FUNCTION_BLOCK TelemetryRelativeHumidities EXTENDS SM_TelemetryRelativeHumidities
VAR_INPUT
END_VAR
VAR_OUTPUT
END_VAR
VAR
    _testVar_TelemetryRelativeHumidities : BOOL;
END_VAR

SUPER^(config := config);

END_FUNCTION_BLOCK

(* stored: Version 1.1.0.1, ProductVersion 3.1.0.36
   POU TelemetryRelativeHumidities: Id {a1d3a85c-8191-4d82-831f-93d259e479d6}, SpecialFunc None *)
